{attribute 'GeneratedUsingTerminal: EL2032-0000-0018'}
{attribute addProperty BoxType "EL2032-0000-0018"}
{attribute addProperty Id "DiagAT %I*BOOL1"}
{attribute addProperty CRC "2804620823"}
{attribute addProperty Size "1"}
TYPE Diag_A72B1E17 :
STRUCT
	{attribute addProperty Name "Diag"}
	Diag AT %I* : BOOL;
END_STRUCT
END_TYPE

(* stored: Version 1.2.0.0, ProductVersion 3.1.4024.9
   DUT Diag_A72B1E17: Id {d8168114-aab2-4bc5-81ec-28e83f86e2e6} *)
